VAR_GLOBAL
  gsPadTitle: STRING;
END_VAR

(* stored: Version 1.1.0.1, ProductVersion 3.1.4024.2
   GVL GVL: Id {b8d203ea-88d0-4d05-99cd-fce0318b441e} *)
